FUNCTION getPercent : INT
VAR_INPUT
    inAct : INT; // actual valuelue
    inMin : INT; // minimum value
    inMax : INT; // maximum possible va
END_VAR
VAR
END_VAR

getPercent := ((inAct - inMin) * 100) / (inMax - inMin);

END_FUNCTION

(* stored: Version 1.1.0.1, ProductVersion 3.1.4024.6
   POU getPercent: Id {d3e00c21-3be2-49a2-9767-12208a2c98d7}, SpecialFunc None *)
